// TwinCAT 3 PLC project Robotino_PLC
// ProgramVersion: 3.1.4022.0
// libraries:
//   Tc2_EtherCAT, * (Beckhoff Automation GmbH)
//   Tc2_MC2, * (Beckhoff Automation GmbH)
//   Tc2_Standard, * (Beckhoff Automation GmbH)
//   Tc2_System, * (Beckhoff Automation GmbH)
//   Tc2_Utilities, * (Beckhoff Automation GmbH)
//   Tc3_Module, * (Beckhoff Automation GmbH)
// project tree:
//   DUTs/ EnumState.TcDUT
//   / PlcTask.TcTTO
//   POUs/COE_Auswertung/ COE_Auswertung.TcPOU, MAIN_COE_Auswertung.TcPOU
//   POUs/Motoransteuerung/ MAIN_Motoransteuerung.TcPOU
//   POUs/Shutdown/ MAIN_Shutdown.TcPOU (not stored), Shutdown.TcPOU
//   POUs/UDP/ MAIN_UDP.TcPOU, UDPConnect.TcPOU (not stored)
// real-time tasks:
//   TASK PLC_Task: cycle T#5ms, priority 2, ADS port 350
//   TASK IrSensor_Task: cycle T#25000us, priority 3, ADS port 351
//   TASK UDP_Task: cycle T#25000us, priority 4, ADS port 354
// motion (NC):
//   TASK Antriebe und Greifer: cycle T#2ms, priority 1, ADS port 501
//   TASK NC-Task 1 SVB: cycle T#10ms, priority 8, ADS port 511
//   AXIS Achse 1 (id 1)
//     Velo: Maximum=1120
//     OtherSettings: AllowMotionCmdToSlave=true
//     encoder EncType=4
//       EncPara: ScaleFactorNumerator=0.00778, MaxCount=#xffffffff
//         Inc: RefMode=2, RefSoftSyncMask=#x0000ffff
//         TimeComp: TimeCompMode=1, EncDelayCycles=4
//     drive DrvType=23
//       Analog: VeloReferenz=942, ScaleFactorActTorque=0.1
//       TimeComp: TaskDelayCycles=1
//     controller CtrType=1
//       CtrPara: PriorControlFactor=1
//         PosDiffControl: Enable=false
//         PID: PosKp=25
//         Observer: BandWidth=20
//   AXIS Achse 2 (id 2)
//     Velo: Maximum=1120
//     OtherSettings: AllowMotionCmdToSlave=true
//     encoder EncType=4
//       EncPara: ScaleFactorNumerator=0.00778, MaxCount=#xffffffff
//         Inc: RefSoftSyncMask=#x0000ffff
//         TimeComp: TimeCompMode=1, EncDelayCycles=4
//     drive DrvType=23
//       Analog: VeloReferenz=942, ScaleFactorActTorque=0.1
//       TimeComp: TaskDelayCycles=1
//     controller CtrType=1
//       CtrPara: PriorControlFactor=1
//         PosDiffControl: Enable=false
//         PID: PosKp=5
//         Observer: BandWidth=20
//   AXIS Achse 3 (id 3)
//     Velo: Maximum=1120
//     OtherSettings: AllowMotionCmdToSlave=true
//     encoder EncType=4
//       EncPara: ScaleFactorNumerator=0.00778, MaxCount=#xffffffff
//         Inc: RefSoftSyncMask=#x0000ffff
//         TimeComp: TimeCompMode=1, EncDelayCycles=4
//     drive DrvType=23
//       Analog: VeloReferenz=942, ScaleFactorActTorque=0.1
//       TimeComp: TaskDelayCycles=1
//     controller CtrType=1
//       CtrPara: PriorControlFactor=1
//         PosDiffControl: Enable=false
//         PID: PosKp=0
//         Observer: BandWidth=20
//   AXIS Achse 4 (id 4)
//     Velo: Maximum=3000
//     OtherSettings: AllowMotionCmdToSlave=true
//     encoder EncType=4
//       EncPara: MaxCount=#x0000ffff
//         Inc: RefSoftSyncMask=#x0000ffff
//     drive DrvType=23
//       Analog: VeloReferenz=3000, ScaleFactorActTorque=0.1
//       TimeComp: TaskDelayCycles=1
//     controller CtrType=1
//       CtrPara: PriorControlFactor=1
//         PosDiffControl: Enable=false
//         Observer: BandWidth=20
// I/O:
//   DEVICE Gerät 1 (EtherCAT), AmsNetId 0.0.0.0.2.1
//     Klemme 1 (EK1200) [EK1200-5000 EtherCAT Netzteil (2A E-Bus)]
//       Motorcontroller 1 [EL7342 2K. DC-Motor-Endstufe (50V, 3.5A)]
//       Motorcontroller 2 [EL7342 2K. DC-Motor-Endstufe (50V, 3.5A)]
//       8 Kanal Digital Input [EL1008 8K. Dig. Eingang 24V, 3ms]
//       4 Kanal Digital Output [EL2004 4K. Dig. Ausgang 24V, 0.5A]
//       8 Kanal Analog Input [EL3068 8K. Ana. Eingang 0-10V]
//       4 Kanal Analog Input [EL3064 4K.Ana. Eingang 0-10V]
//       Netzteilklemme 5V [EL9505 Netzteilklemme 5V]
//       Klemme 9 (EL9011) [EL9011 Endklemme]
//   DEVICE WLAN Adapter
// variable links:
//   Device 1 (EtherCAT) <-> irSensors/irSensors_Obj1 (updateIrSensors)
//     Term 1 (EK1200)/4 Kanal Analog Input/AI Standard Channel 1/IR Sensor 9 <-> Inputs/irInputData[8]
//     Term 1 (EK1200)/8 Kanal Analog Input/AI Standard Channel 1/IR Sensor 1 <-> Inputs/irInputData[0]
//     Term 1 (EK1200)/8 Kanal Analog Input/AI Standard Channel 2/IR Sensor 2 <-> Inputs/irInputData[1]
//     Term 1 (EK1200)/8 Kanal Analog Input/AI Standard Channel 3/IR Sensor 3 <-> Inputs/irInputData[2]
//     Term 1 (EK1200)/8 Kanal Analog Input/AI Standard Channel 4/IR Sensor 4 <-> Inputs/irInputData[3]
//     Term 1 (EK1200)/8 Kanal Analog Input/AI Standard Channel 5/IR Sensor 5 <-> Inputs/irInputData[4]
//     Term 1 (EK1200)/8 Kanal Analog Input/AI Standard Channel 6/IR Sensor 6 <-> Inputs/irInputData[5]
//     Term 1 (EK1200)/8 Kanal Analog Input/AI Standard Channel 7/IR Sensor 7 <-> Inputs/irInputData[6]
//     Term 1 (EK1200)/8 Kanal Analog Input/AI Standard Channel 8/IR Sensor 8 <-> Inputs/irInputData[7]
//   Antriebe und Greifer/Axes/Achse 1 <-> Device 1 (EtherCAT)/Term 1 (EK1200)/Motorcontroller 2
//     Drive/Inputs/In/nState1 @bit 3 <-> DCM Status Channel 1/Status/Error
//     Drive/Inputs/In/nState1 @bit 5 <-> DCM Status Channel 1/Status/Moving negative
//     Drive/Inputs/In/nState1 @bit 4 <-> DCM Status Channel 1/Status/Moving positive
//     Drive/Inputs/In/nState1 @bit 1 <-> DCM Status Channel 1/Status/Ready
//     Drive/Inputs/In/nState1 <-> DCM Status Channel 1/Status/Ready to enable
//     Drive/Inputs/In/nState1 @bit 6 <-> DCM Status Channel 1/Status/Torque reduced
//     Drive/Inputs/In/nState1 @bit 2 <-> DCM Status Channel 1/Status/Warning
//     Drive/Inputs/In/nState2 @bit 3 <-> DCM Status Channel 1/Status/Digital input 1
//     Drive/Inputs/In/nState2 @bit 4 <-> DCM Status Channel 1/Status/Digital input 2
//     Drive/Inputs/In/nState2 @bit 5 <-> DCM Status Channel 1/Status/Sync error
//     Drive/Inputs/In/nState2 @bit 7 <-> DCM Status Channel 1/Status/TxPDO Toggle
//     Drive/Inputs/In/nState4 @bit 1 <-> WcState/InputToggle
//     Drive/Inputs/In/nState4 <-> WcState/WcState
//     Drive/Outputs/Out/nCtrl1 <-> DCM Control Channel 1/Control/Enable
//     Drive/Outputs/Out/nCtrl1 @bit 2 <-> DCM Control Channel 1/Control/Reduce torque
//     Drive/Outputs/Out/nCtrl1 @bit 1 <-> DCM Control Channel 1/Control/Reset
//     Drive/Outputs/Out/nDataOut2[0] <-> DCM Velocity Channel 1/Velocity
//     Enc/Inputs/In/nDataIn1 <-> ENC Status Channel 1/Counter value
//     Enc/Inputs/In/nDataIn2 <-> ENC Status Channel 1/Latch value
//     Enc/Inputs/In/nState1 @bit 4 <-> ENC Status Channel 1/Status/Counter overflow
//     Enc/Inputs/In/nState1 @bit 3 <-> ENC Status Channel 1/Status/Counter underflow
//     Enc/Inputs/In/nState1 @bit 7 <-> ENC Status Channel 1/Status/Extrapolation stall
//     Enc/Inputs/In/nState1 @bit 1 <-> ENC Status Channel 1/Status/Latch extern valid
//     Enc/Inputs/In/nState1 @bit 2 <-> ENC Status Channel 1/Status/Set counter done
//     Enc/Inputs/In/nState2 @bit 4 <-> ENC Status Channel 1/Status/Status of extern latch
//     Enc/Inputs/In/nState2 <-> ENC Status Channel 1/Status/Status of input A
//     Enc/Inputs/In/nState2 @bit 1 <-> ENC Status Channel 1/Status/Status of input B
//     Enc/Inputs/In/nState2 @bit 5 <-> ENC Status Channel 1/Status/Sync error
//     Enc/Inputs/In/nState2 @bit 7 <-> ENC Status Channel 1/Status/TxPDO Toggle
//     Enc/Inputs/In/nState4 @bit 1 <-> WcState/InputToggle
//     Enc/Inputs/In/nState4 <-> WcState/WcState
//     Enc/Outputs/Out/nCtrl1 @bit 3 <-> ENC Control Channel 1/Control/Enable latch extern on negative edge
//     Enc/Outputs/Out/nCtrl1 @bit 1 <-> ENC Control Channel 1/Control/Enable latch extern on positive edge
//     Enc/Outputs/Out/nCtrl1 @bit 2 <-> ENC Control Channel 1/Control/Set counter
//     Enc/Outputs/Out/nDataOut1 <-> ENC Control Channel 1/Set counter value
//   Antriebe und Greifer/Axes/Achse 1 <-> velocityConverterToCartesian/velocityConverterToCartesian_Obj
//     Outputs/ToPlc/ActVelo <-> Inputs/velocityFromMotor1
//   Antriebe und Greifer/Axes/Achse 2 <-> Device 1 (EtherCAT)/Term 1 (EK1200)/Motorcontroller 1
//     Drive/Inputs/In/nState1 @bit 3 <-> DCM Status Channel 2/Status/Error
//     Drive/Inputs/In/nState1 @bit 5 <-> DCM Status Channel 2/Status/Moving negative
//     Drive/Inputs/In/nState1 @bit 4 <-> DCM Status Channel 2/Status/Moving positive
//     Drive/Inputs/In/nState1 @bit 1 <-> DCM Status Channel 2/Status/Ready
//     Drive/Inputs/In/nState1 <-> DCM Status Channel 2/Status/Ready to enable
//     Drive/Inputs/In/nState1 @bit 6 <-> DCM Status Channel 2/Status/Torque reduced
//     Drive/Inputs/In/nState1 @bit 2 <-> DCM Status Channel 2/Status/Warning
//     Drive/Inputs/In/nState2 @bit 3 <-> DCM Status Channel 2/Status/Digital input 1
//     Drive/Inputs/In/nState2 @bit 4 <-> DCM Status Channel 2/Status/Digital input 2
//     Drive/Inputs/In/nState2 @bit 5 <-> DCM Status Channel 2/Status/Sync error
//     Drive/Inputs/In/nState2 @bit 7 <-> DCM Status Channel 2/Status/TxPDO Toggle
//     Drive/Inputs/In/nState4 @bit 1 <-> WcState/InputToggle
//     Drive/Inputs/In/nState4 <-> WcState/WcState
//     Drive/Outputs/Out/nCtrl1 <-> DCM Control Channel 2/Control/Enable
//     Drive/Outputs/Out/nCtrl1 @bit 2 <-> DCM Control Channel 2/Control/Reduce torque
//     Drive/Outputs/Out/nCtrl1 @bit 1 <-> DCM Control Channel 2/Control/Reset
//     Drive/Outputs/Out/nDataOut2[0] <-> DCM Velocity Channel 2/Velocity
//     Enc/Inputs/In/nDataIn1 <-> ENC Status Channel 2/Counter value
//     Enc/Inputs/In/nDataIn2 <-> ENC Status Channel 2/Latch value
//     Enc/Inputs/In/nState1 @bit 4 <-> ENC Status Channel 2/Status/Counter overflow
//     Enc/Inputs/In/nState1 @bit 3 <-> ENC Status Channel 2/Status/Counter underflow
//     Enc/Inputs/In/nState1 @bit 7 <-> ENC Status Channel 2/Status/Extrapolation stall
//     Enc/Inputs/In/nState1 @bit 1 <-> ENC Status Channel 2/Status/Latch extern valid
//     Enc/Inputs/In/nState1 @bit 2 <-> ENC Status Channel 2/Status/Set counter done
//     Enc/Inputs/In/nState2 @bit 4 <-> ENC Status Channel 2/Status/Status of extern latch
//     Enc/Inputs/In/nState2 <-> ENC Status Channel 2/Status/Status of input A
//     Enc/Inputs/In/nState2 @bit 1 <-> ENC Status Channel 2/Status/Status of input B
//     Enc/Inputs/In/nState2 @bit 5 <-> ENC Status Channel 2/Status/Sync error
//     Enc/Inputs/In/nState2 @bit 7 <-> ENC Status Channel 2/Status/TxPDO Toggle
//     Enc/Inputs/In/nState4 @bit 1 <-> WcState/InputToggle
//     Enc/Inputs/In/nState4 <-> WcState/WcState
//     Enc/Outputs/Out/nCtrl1 @bit 3 <-> ENC Control Channel 2/Control/Enable latch extern on negative edge
//     Enc/Outputs/Out/nCtrl1 @bit 1 <-> ENC Control Channel 2/Control/Enable latch extern on positive edge
//     Enc/Outputs/Out/nCtrl1 @bit 2 <-> ENC Control Channel 2/Control/Set counter
//     Enc/Outputs/Out/nDataOut1 <-> ENC Control Channel 2/Set counter value
//   Antriebe und Greifer/Axes/Achse 2 <-> velocityConverterToCartesian/velocityConverterToCartesian_Obj
//     Outputs/ToPlc/ActVelo <-> Inputs/velocityFromMotor2
//   Antriebe und Greifer/Axes/Achse 3 <-> Device 1 (EtherCAT)/Term 1 (EK1200)/Motorcontroller 1
//     Drive/Inputs/In/nState1 @bit 3 <-> DCM Status Channel 1/Status/Error
//     Drive/Inputs/In/nState1 @bit 5 <-> DCM Status Channel 1/Status/Moving negative
//     Drive/Inputs/In/nState1 @bit 4 <-> DCM Status Channel 1/Status/Moving positive
//     Drive/Inputs/In/nState1 @bit 1 <-> DCM Status Channel 1/Status/Ready
//     Drive/Inputs/In/nState1 <-> DCM Status Channel 1/Status/Ready to enable
//     Drive/Inputs/In/nState1 @bit 6 <-> DCM Status Channel 1/Status/Torque reduced
//     Drive/Inputs/In/nState1 @bit 2 <-> DCM Status Channel 1/Status/Warning
//     Drive/Inputs/In/nState2 @bit 3 <-> DCM Status Channel 1/Status/Digital input 1
//     Drive/Inputs/In/nState2 @bit 4 <-> DCM Status Channel 1/Status/Digital input 2
//     Drive/Inputs/In/nState2 @bit 5 <-> DCM Status Channel 1/Status/Sync error
//     Drive/Inputs/In/nState2 @bit 7 <-> DCM Status Channel 1/Status/TxPDO Toggle
//     Drive/Inputs/In/nState4 @bit 1 <-> WcState/InputToggle
//     Drive/Inputs/In/nState4 <-> WcState/WcState
//     Drive/Outputs/Out/nCtrl1 <-> DCM Control Channel 1/Control/Enable
//     Drive/Outputs/Out/nCtrl1 @bit 2 <-> DCM Control Channel 1/Control/Reduce torque
//     Drive/Outputs/Out/nCtrl1 @bit 1 <-> DCM Control Channel 1/Control/Reset
//     Drive/Outputs/Out/nDataOut2[0] <-> DCM Velocity Channel 1/Velocity
//     Enc/Inputs/In/nDataIn1 <-> ENC Status Channel 1/Counter value
//     Enc/Inputs/In/nDataIn2 <-> ENC Status Channel 1/Latch value
//     Enc/Inputs/In/nState1 @bit 4 <-> ENC Status Channel 1/Status/Counter overflow
//     Enc/Inputs/In/nState1 @bit 3 <-> ENC Status Channel 1/Status/Counter underflow
//     Enc/Inputs/In/nState1 @bit 7 <-> ENC Status Channel 1/Status/Extrapolation stall
//     Enc/Inputs/In/nState1 @bit 1 <-> ENC Status Channel 1/Status/Latch extern valid
//     Enc/Inputs/In/nState1 @bit 2 <-> ENC Status Channel 1/Status/Set counter done
//     Enc/Inputs/In/nState2 @bit 4 <-> ENC Status Channel 1/Status/Status of extern latch
//     Enc/Inputs/In/nState2 <-> ENC Status Channel 1/Status/Status of input A
//     Enc/Inputs/In/nState2 @bit 1 <-> ENC Status Channel 1/Status/Status of input B
//     Enc/Inputs/In/nState2 @bit 5 <-> ENC Status Channel 1/Status/Sync error
//     Enc/Inputs/In/nState2 @bit 7 <-> ENC Status Channel 1/Status/TxPDO Toggle
//     Enc/Inputs/In/nState4 @bit 1 <-> WcState/InputToggle
//     Enc/Inputs/In/nState4 <-> WcState/WcState
//     Enc/Outputs/Out/nCtrl1 @bit 3 <-> ENC Control Channel 1/Control/Enable latch extern on negative edge
//     Enc/Outputs/Out/nCtrl1 @bit 1 <-> ENC Control Channel 1/Control/Enable latch extern on positive edge
//     Enc/Outputs/Out/nCtrl1 @bit 2 <-> ENC Control Channel 1/Control/Set counter
//     Enc/Outputs/Out/nDataOut1 <-> ENC Control Channel 1/Set counter value
//   Antriebe und Greifer/Axes/Achse 3 <-> velocityConverterToCartesian/velocityConverterToCartesian_Obj
//     Outputs/ToPlc/ActVelo <-> Inputs/velocityFromMotor3
//   Antriebe und Greifer/Axes/Achse 4 <-> Device 1 (EtherCAT)/Term 1 (EK1200)/Motorcontroller 2
//     Drive/Inputs/In/nState1 @bit 3 <-> DCM Status Channel 2/Status/Error
//     Drive/Inputs/In/nState1 @bit 5 <-> DCM Status Channel 2/Status/Moving negative
//     Drive/Inputs/In/nState1 @bit 4 <-> DCM Status Channel 2/Status/Moving positive
//     Drive/Inputs/In/nState1 @bit 1 <-> DCM Status Channel 2/Status/Ready
//     Drive/Inputs/In/nState1 <-> DCM Status Channel 2/Status/Ready to enable
//     Drive/Inputs/In/nState1 @bit 6 <-> DCM Status Channel 2/Status/Torque reduced
//     Drive/Inputs/In/nState1 @bit 2 <-> DCM Status Channel 2/Status/Warning
//     Drive/Inputs/In/nState2 @bit 3 <-> DCM Status Channel 2/Status/Digital input 1
//     Drive/Inputs/In/nState2 @bit 4 <-> DCM Status Channel 2/Status/Digital input 2
//     Drive/Inputs/In/nState2 @bit 5 <-> DCM Status Channel 2/Status/Sync error
//     Drive/Inputs/In/nState2 @bit 7 <-> DCM Status Channel 2/Status/TxPDO Toggle
//     Drive/Inputs/In/nState4 @bit 1 <-> WcState/InputToggle
//     Drive/Inputs/In/nState4 <-> WcState/WcState
//     Drive/Outputs/Out/nCtrl1 <-> DCM Control Channel 2/Control/Enable
//     Drive/Outputs/Out/nCtrl1 @bit 2 <-> DCM Control Channel 2/Control/Reduce torque
//     Drive/Outputs/Out/nCtrl1 @bit 1 <-> DCM Control Channel 2/Control/Reset
//     Drive/Outputs/Out/nDataOut2[0] <-> DCM Velocity Channel 2/Velocity
//     Enc/Inputs/In/nState4 @bit 1 <-> WcState/InputToggle
//     Enc/Inputs/In/nState4 <-> WcState/WcState
//   Robotino_PLC/Robotino_PLC Instance <-> Device 1 (EtherCAT)/Term 1 (EK1200)/8 Kanal Digital Input
//     PlcTask Inputs/MAIN_Motoransteuerung.bumper <-> Channel 2/Bumper Sensor
//     PlcTask Inputs/Shutdown.bStart <-> Channel 8/Shutdown
//   Robotino_PLC/Robotino_PLC Instance <-> Antriebe und Greifer/Axes/Achse 1
//     PlcTask Inputs/MAIN_Motoransteuerung.axis1.NcToPlc <-> Outputs/ToPlc
//     PlcTask Outputs/MAIN_Motoransteuerung.axis1.PlcToNc <-> Inputs/FromPlc
//   Robotino_PLC/Robotino_PLC Instance <-> Antriebe und Greifer/Axes/Achse 2
//     PlcTask Inputs/MAIN_Motoransteuerung.axis2.NcToPlc <-> Outputs/ToPlc
//     PlcTask Outputs/MAIN_Motoransteuerung.axis2.PlcToNc <-> Inputs/FromPlc
//   Robotino_PLC/Robotino_PLC Instance <-> Antriebe und Greifer/Axes/Achse 3
//     PlcTask Inputs/MAIN_Motoransteuerung.axis3.NcToPlc <-> Outputs/ToPlc
//     PlcTask Outputs/MAIN_Motoransteuerung.axis3.PlcToNc <-> Inputs/FromPlc
//   Robotino_PLC/Robotino_PLC Instance <-> velocityConverterToMotors/velocityConverterToMotors_Obj
//     PlcTask Inputs/MAIN_Motoransteuerung.directionToMotors1 <-> Outputs/directionToMotors1
//     PlcTask Inputs/MAIN_Motoransteuerung.directionToMotors2 <-> Outputs/directionToMotors2
//     PlcTask Inputs/MAIN_Motoransteuerung.directionToMotors3 <-> Outputs/directionToMotors3
//     PlcTask Inputs/MAIN_Motoransteuerung.velocityToMotors1 <-> Outputs/velocityToMotors1
//     PlcTask Inputs/MAIN_Motoransteuerung.velocityToMotors2 <-> Outputs/velocityToMotors2
//     PlcTask Inputs/MAIN_Motoransteuerung.velocityToMotors3 <-> Outputs/velocityToMotors3

CONFIGURATION Robotino_PLC
    RESOURCE PLC ON TwinCAT3
        TASK PlcTask(INTERVAL := T#5ms, PRIORITY := 2);
        PROGRAM MAIN_Motoransteuerung WITH PlcTask : MAIN_Motoransteuerung;
        PROGRAM MAIN_Shutdown WITH PlcTask : MAIN_Shutdown;
        PROGRAM MAIN_UDP WITH PlcTask : MAIN_UDP;
        PROGRAM MAIN_COE_Auswertung WITH PlcTask : MAIN_COE_Auswertung;
    END_RESOURCE
END_CONFIGURATION

// ---- DUTs/EnumState.TcDUT
{attribute 'qualified_only'}
{attribute 'strict'}
TYPE EnumState :
(
	init,
	drive1,
	drive2,
	reset
);
END_TYPE

// ---- POUs/Motoransteuerung/MAIN_Motoransteuerung.TcPOU
PROGRAM MAIN_Motoransteuerung
VAR
	//Achsen Referenzen
	axis1: AXIS_REF;
	axis2: AXIS_REF;
	axis3: AXIS_REF;
	
	//Objekte um Achsen anzusteuern
	powerAxis1: MC_Power;
	driveAxis1: MC_MoveVelocity;
	driveAxis12: MC_MoveVelocity;
	resetAxis1: MC_Reset;
	
	powerAxis2: MC_Power;
	driveAxis2: MC_MoveVelocity;
	driveAxis22: MC_MoveVelocity;
	resetAxis2: MC_Reset;
	
	powerAxis3: MC_Power;
	driveAxis3: MC_MoveVelocity;
	driveAxis32: MC_MoveVelocity;
	resetAxis3: MC_Reset;
	
	//Achse Freischalten, Regler Freischalten
	enableControl: BOOL	:=0;
	enablePos: BOOL		:=0;
	enableNeg: BOOL		:=0;
	override:  LREAL	:=0;
	
	//Fahrbefehl Ausführen
	driveExecute: BOOL	:=0;
	
	//State Maschine
	nextState:EnumState	:=EnumState.init;
	state:EnumState		:=EnumState.init;
	switchDrive:INT		:=0;
	
	//Umgerechnete Werte
	vX:		LREAL:=0;
	vY:		LREAL:=0;
	vTheta:	LREAL:=0;
	v0:		LREAL:=0;
	v1:		LREAL:=0;
	v2:		LREAL:=0;
	
	//Fahrbefehle für Motor MC_DRIVEVELOCITY
	velocityToMotor1: LREAL:=0;
	velocityToMotor2: LREAL:=0;
	velocityToMotor3: LREAL:=0;
	directionToMotor1: INT:=0;
	directionToMotor2: INT:=0;
	directionToMotor3: INT:=0;
	
	// Skalierung auf maximale Geschwindigkeit
	vMax:LREAL:=942;
	velocityToMotorsTf:LREAL:=0;
	
	//Inputs: CartesianToMotors + Bumper
	
	vXCartesianToMotors 	AT%I*:LREAL:=0;
	vYCartesianToMotors 	AT%I*:LREAL:=0;
	vThetaCartesianToMotors AT%I*:LREAL:=0;
	
	bumper	   AT%I*: BOOL:=0;
END_VAR

axis1.ReadStatus();
axis2.ReadStatus();
axis3.ReadStatus();

// Konverzierung ToMotors Anfang********************************************************

//	  conversion from positive and / or negative longitudinal, lateral and
//	  rotational velocities(in milimeters per second) to three separate
//	  positive motor velocities(resolution: 1Byte) and their rotation
//    direction
//inputs:  	velocityX (longitudinal velocity in milimeters per second)
//         	velocityY (lateral velocity in milimeters per second)
//			theta     (rotational velocity in milimeters per second)
//outputs : velocityMotor0	
//			velocityMotor1
//			velocityMotor2
//		directionMotor0 (rotating direction of motor1, 1 := positiveDirection, 3 := negartiveDirection)
//		directionMotor1 (rotating direction of motor2, 1 := positiveDirection, 3 := negartiveDirection)
//		directionMotor2 (rotating direction of motor3, 1 := positiveDirection, 3 := negartiveDirection)
//conversion from longitudinal, lateral & rotational velocity to the
//three separate motor velocities

//Maximal Speed
//IF 	vXCartesianToMotors > 500 	THEN
//	vX := 500;
  
//	vX := vXCartesianToMotors;
//END_IF

//IF	vYCartesianToMotors > 500	THEN
//	vY := 500;
//ELSIF vYCartesianToMotors < -500 THEN
//	vY := -500;
//ELSE
//	vY :=vYCartesianToMotors;
//END_IF
	
//IF vThetaCartesianToMotors > 3.14 THEN
//	vTheta:=3.14;
//ELSIF vThetaCartesianToMotors < -3.14 THEN
//	vTheta:=-3.14;	
//ELSE
//	vTheta:= vThetaCartesianToMotors;
//END_IF

vX:=vXCartesianToMotors;
vY:=vYCartesianToMotors;
vTheta:=vThetaCartesianToMotors;

v0 := (-vX * COS(30.0*PI/180))	+ (vY * COS(60.0*PI/180))	+ (vTheta * 135.0);
v1 := 0.0						+ (-vY)						+ (vTheta * 135.0);
v2 := (vX * COS(30.0*PI/180))	+ (vY * COS(60.0*PI/180))	+ (vTheta * 135.0);
	
//division OF motor velocities into absolute velocity AND rotating
//direction
IF v0 < 0 THEN
	directionToMotor1 := 1;
	velocityToMotor1 := -v0;
ELSE
	directionToMotor1:= 3;
	velocityToMotor1:= v0;
END_IF

IF v1 < 0 THEN
	directionToMotor2:= 1;
	velocityToMotor2:= -v1;
ELSE
	directionToMotor2:= 3;
	velocityToMotor2:= v1;
END_IF

IF(v2 < 0)THEN
	directionToMotor3 := 1;
	velocityToMotor3  := -v2;
ELSE
	directionToMotor3 := 3;
	velocityToMotor3  := v2;
END_IF


IF velocityToMotor1 > vMax THEN
    velocityToMotorsTf:= velocityToMotor1;
    
    velocityToMotor1:= vMax;
    velocityToMotor2:= vMax * velocityToMotor2 / velocityToMotorsTf;
    velocityToMotor3:= vMax * velocityToMotor3 / velocityToMotorsTf;
END_IF

IF velocityToMotor2 > vMax THEN
    velocityToMotorsTf:= velocityToMotor2;
    
    velocityToMotor1:= vMax * velocityToMotor1 / velocityToMotorsTf;
    velocityToMotor2:= vMax;
    velocityToMotor3:= vMax * velocityToMotor3 / velocityToMotorsTf;
END_IF

IF velocityToMotor3 > vMax THEN
    velocityToMotorsTf:= velocityToMotor3;
    
    velocityToMotor1:= vMax * velocityToMotor1 / velocityToMotorsTf;
    velocityToMotor2:= vMax * velocityToMotor2 / velocityToMotorsTf;
    velocityToMotor3:= vMax;
END_IF
// Konverzierung ToMotors ENDE********************************************************


//START STATE MACHINE MOTORANSTEUERUNG
CASE state OF
	EnumState.init:
		enableControl:=1;
		enablePos:=1;
		enableNeg:=1;
		override:=100;
		
		powerAxis1(Axis:=axis1,Enable:=enableControl,Enable_Positive:=enablePos,Enable_Negative:=enableNeg,Override:=override);
		powerAxis2(Axis:=axis2,Enable:=enableControl,Enable_Positive:=enablePos,Enable_Negative:=enableNeg,Override:=override);
		powerAxis3(Axis:=axis3,Enable:=enableControl,Enable_Positive:=enablePos,Enable_Negative:=enableNeg,Override:=override);
		IF (powerAxis1.Status AND powerAxis2.Status AND powerAxis3.Status) THEN	
			nextState:=EnumState.drive1; 
			driveExecute:=1;
		END_IF
		IF (powerAxis1.Error OR powerAxis2.Error OR powerAxis3.Error) THEN
			nextState:=EnumState.reset;
		END_IF
		
	EnumState.drive1:
	
		driveAxis1(Axis:=axis1,Velocity:=velocityToMotor1,Direction:=directionToMotor1,Execute:=driveExecute,BufferMode:=MC_Aborting);
		driveAxis2(Axis:=axis2,Velocity:=velocityToMotor2,Direction:=directionToMotor2,Execute:=driveExecute,BufferMode:=MC_Aborting);
		driveAxis3(Axis:=axis3,Velocity:=velocityToMotor3,Direction:=directionToMotor3,Execute:=driveExecute,BufferMode:=MC_Aborting);
		switchDrive:=switchDrive+1;
		
		IF (switchDrive=2) THEN
			switchDrive:=0;
			nextState:=EnumState.drive2;
			driveExecute:=0;
			driveAxis1(Axis:=axis1,Execute:=driveExecute);
			driveAxis2(Axis:=axis2,Execute:=driveExecute);
			driveAxis3(Axis:=axis3,Execute:=driveExecute);
			driveExecute:=1;
		END_IF
		
		IF (powerAxis1.Error OR powerAxis2.Error OR powerAxis3.Error) THEN
			nextState:=EnumState.reset;
		END_IF
		
	EnumState.drive2:
	
		driveAxis1(Axis:=axis1,Velocity:=velocityToMotor1,Direction:=directionToMotor1,Execute:=driveExecute,BufferMode:=MC_Aborting);
		driveAxis2(Axis:=axis2,Velocity:=velocityToMotor2,Direction:=directionToMotor2,Execute:=driveExecute,BufferMode:=MC_Aborting);
		driveAxis3(Axis:=axis3,Velocity:=velocityToMotor3,Direction:=directionToMotor3,Execute:=driveExecute,BufferMode:=MC_Aborting);
		switchDrive:=switchDrive+1;
		
		IF (switchDrive=2) THEN
			switchDrive:=0;
			nextState:=EnumState.drive1;
			driveExecute:=0;
			driveAxis1(Axis:=axis1,Execute:=driveExecute);
			driveAxis2(Axis:=axis2,Execute:=driveExecute);
			driveAxis3(Axis:=axis3,Execute:=driveExecute);
			driveExecute:=1;
		END_IF
		IF (powerAxis1.Error OR powerAxis2.Error OR powerAxis3.Error OR bumper) THEN
			nextState:=EnumState.reset;
		END_IF	
	EnumState.reset:
	
		powerAxis1(Axis:=axis1,Enable:=0,Enable_Positive:=0,Enable_Negative:=0,Override:=0);
		powerAxis2(Axis:=axis1,Enable:=0,Enable_Positive:=0,Enable_Negative:=0,Override:=0);
		powerAxis3(Axis:=axis1,Enable:=0,Enable_Positive:=0,Enable_Negative:=0,Override:=0);
		driveAxis1(Axis:=axis1,Velocity:=0,Direction:=0,Execute:=0,BufferMode:=MC_Aborting);
		driveAxis2(Axis:=axis1,Velocity:=0,Direction:=0,Execute:=0,BufferMode:=MC_Aborting);
		driveAxis3(Axis:=axis1,Velocity:=0,Direction:=0,Execute:=0,BufferMode:=MC_Aborting);
	
		resetAxis1(Axis:=axis1,Execute:=1);
		resetAxis2(Axis:=axis2,Execute:=1);
		resetAxis3(Axis:=axis3,Execute:=1);
	
		IF (resetAxis1.Done AND resetAxis2.Done AND resetAxis3.Done) THEN
					;
				END_IF	
	ELSE
		nextState:=EnumState.reset;
END_CASE
state:=nextState;

END_PROGRAM

// ---- POUs/UDP/MAIN_UDP.TcPOU
PROGRAM MAIN_UDP
VAR
	//sPaketinhalt	: LREAL;
	//nPaketlaenge	: UDINT;
	
	x	  AT%Q*	: ARRAY[1..4] OF LREAL;
	y	  AT%Q*	: ARRAY[1..4] OF LREAL;
	theta AT%Q*	: ARRAY[1..4] OF LREAL;
	udp1 : UDPConnect;
END_VAR

udp1();

END_PROGRAM

// ---- POUs/COE_Auswertung/MAIN_COE_Auswertung.TcPOU
PROGRAM MAIN_COE_Auswertung
VAR
	COE_Auswertung_0: TwinCAT_Device.Robotino_PLC.COE_Auswertung;
END_VAR

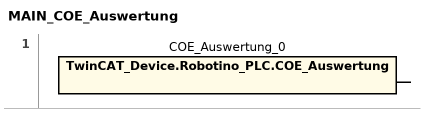
// NETWORK 1
COE_Auswertung_0(); // TwinCAT_Device.Robotino_PLC.COE_Auswertung

END_PROGRAM

// ---- POUs/COE_Auswertung/COE_Auswertung.TcPOU
FUNCTION_BLOCK COE_Auswertung
VAR_INPUT
END_VAR
VAR_OUTPUT
END_VAR
VAR
	MotorstromAchse1: FB_EcCoESdoRead;
	Achse1Motorspannung: LREAL;
	Achse2Motorspannung: LREAL;
	Achse3Motorspannung: LREAL;
	
	Achse1Motorstrom: LREAL;
	Achse2Motorstrom: LREAL;
	Achse3Motorstrom: LREAL;
	
	MotorspannungAchse1: FB_EcCoESdoRead;
	MotorstromAchse2: FB_EcCoESdoRead;
	MotorspannungAchse2: FB_EcCoESdoRead;
	MotorspannungAchse3: FB_EcCoESdoRead;
	MotorstromAchse3: FB_EcCoESdoRead;
END_VAR

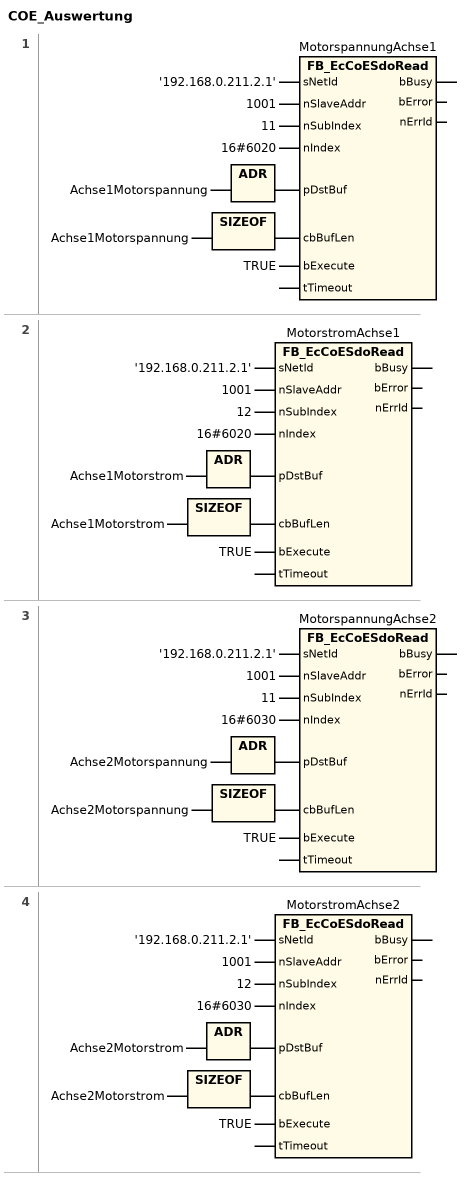
// NETWORK 1
MotorspannungAchse1(
    sNetId := '192.168.0.211.2.1',
    nSlaveAddr := 1001,
    nSubIndex := 11,
    nIndex := 16#6020,
    pDstBuf := ADR(Achse1Motorspannung),
    cbBufLen := SIZEOF(Achse1Motorspannung),
    bExecute := TRUE); // FB_EcCoESdoRead

// NETWORK 2
MotorstromAchse1(
    sNetId := '192.168.0.211.2.1',
    nSlaveAddr := 1001,
    nSubIndex := 12,
    nIndex := 16#6020,
    pDstBuf := ADR(Achse1Motorstrom),
    cbBufLen := SIZEOF(Achse1Motorstrom),
    bExecute := TRUE); // FB_EcCoESdoRead

// NETWORK 3
MotorspannungAchse2(
    sNetId := '192.168.0.211.2.1',
    nSlaveAddr := 1001,
    nSubIndex := 11,
    nIndex := 16#6030,
    pDstBuf := ADR(Achse2Motorspannung),
    cbBufLen := SIZEOF(Achse2Motorspannung),
    bExecute := TRUE); // FB_EcCoESdoRead

// NETWORK 4
MotorstromAchse2(
    sNetId := '192.168.0.211.2.1',
    nSlaveAddr := 1001,
    nSubIndex := 12,
    nIndex := 16#6030,
    pDstBuf := ADR(Achse2Motorstrom),
    cbBufLen := SIZEOF(Achse2Motorstrom),
    bExecute := TRUE); // FB_EcCoESdoRead

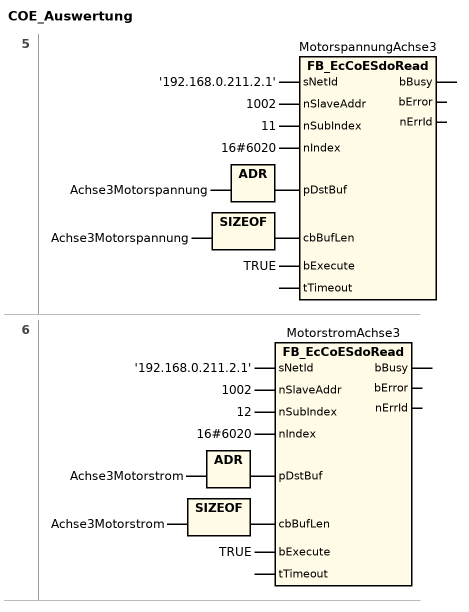
// NETWORK 5
MotorspannungAchse3(
    sNetId := '192.168.0.211.2.1',
    nSlaveAddr := 1002,
    nSubIndex := 11,
    nIndex := 16#6020,
    pDstBuf := ADR(Achse3Motorspannung),
    cbBufLen := SIZEOF(Achse3Motorspannung),
    bExecute := TRUE); // FB_EcCoESdoRead

// NETWORK 6
MotorstromAchse3(
    sNetId := '192.168.0.211.2.1',
    nSlaveAddr := 1002,
    nSubIndex := 12,
    nIndex := 16#6020,
    pDstBuf := ADR(Achse3Motorstrom),
    cbBufLen := SIZEOF(Achse3Motorstrom),
    bExecute := TRUE); // FB_EcCoESdoRead

END_FUNCTION_BLOCK

// ---- POUs/Shutdown/Shutdown.TcPOU
PROGRAM Shutdown
VAR
	bStart	AT%I* : BOOL := FALSE;
	Shutdown_Block: NT_Shutdown;
END_VAR

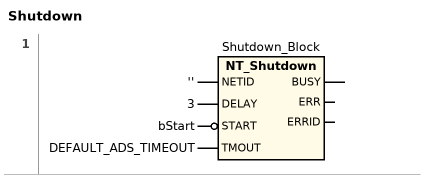
// NETWORK 1
Shutdown_Block(NETID := '', DELAY := 3, START := NOT bStart, TMOUT := DEFAULT_ADS_TIMEOUT); // NT_Shutdown

END_PROGRAM
